Staubli VAL3: setFrameId.pgx

public program setFrameId(num x_nIndex)
begin
  // set the Frame
  jEditPoint.nIndexFrame=x_nIndex
end
